(* CODESYS project emCoSys, 3.3.1.1 (IMACS GmbH).library
   Description: Driver for connecting an emBRICK®-LocalMaster via TCP/IP or RS485 over the Modbus LargeBlock Protokoll.
   Author: IMACS GmbH
   Version: 3.3.1.1
   CompiledLibraryCompatibilityVersion: CODESYS V3.5 SP16 Patch 4
   Company: IMACS GmbH
   Title: emCoSys
   LanguageModelAttribute: qualified-access-only
   DefaultNamespace: TPL

Project tree, tasks and I/O mapping:
  CODESYS_Control_Win_V3 : CODESYS Control Win V3, 3S - Smart Software Solutions GmbH, version 3.5.16.40
    application Application
      libraries: SysCom, 3.5.15.0 (System); SysTypes2 Interfaces, * (System)
  libraries: SysMem, * (System); SysCpuHandling, * (System); IoDrvBase, * (System); IoStandard, * (System); IoDriver Parameter Interfaces, * (System); Base Interfaces, * (System); IoDriver Interfaces, * (System); BASIC, 3.31 (OSCAT); CAA Memory, 3.5.12.0 (CAA Technical Workgroup); CAA Types Extern, 3.5.13.0 (CAA Technical Workgroup); Standard, 3.5.15.0 (System); SysSocket, 3.5.15.0 (System); CAA SerialCom, 3.5.15.0 (CAA Technical Workgroup); SysTypes2 Interfaces, * (System); CmpErrors2 Interfaces, * (System)
  function block emCoSys [ST]: IoDrvWriteParameter, IoDrvReadParameter, IoDrvReadInputs, IoDrvIdentify, IoDrvUpdateConfiguration, IoDrvWatchdogTrigger, IoDrvScanModules, IoDrvUpdateMapping, IoDrvWriteOutputs, IoDrvStartBusCycle, IoDrvGetModuleDiagnosis, QueryInterface, FB_Reinit, Initialize, FB_Exit, FB_Init, IoDrvGetConnector, init, connecting, connectionTimedOut, sendInitRq, recvInitRq, receiveData, sendData, closeSocket, initConnection, GetInitializationData, getVars, CRCModbus
  data type emBRICKData
  data type emBRICKMaster
  data type emBRICKSlave
  data type STATES
  data type COM_TYPES
*)

// emBRICKData
TYPE emBRICKData :
STRUCT
	numOfSlaves : BYTE := 0;
	slaves : ARRAY[0..31] OF emBRICKSlave;
	master : emBRICKMaster;
	localMasterAddress : STRING;
	localMasterPort : UINT;
	pRxData : POINTER TO ARRAY[0..252] OF BYTE;
	pTxData : POINTER TO ARRAY[0..252] OF BYTE;
END_STRUCT
END_TYPE

// emBRICKMaster
TYPE emBRICKMaster :
STRUCT
	ID : WORD := 0;
	protocolVersion : BYTE := 0;
	version : BYTE := 0;
	masterType : BYTE := 0;
	uartType : WORD := 0;	
END_STRUCT
END_TYPE

// emBRICKSlave
TYPE emBRICKSlave :
STRUCT
	status : BYTE := 0;
	dataLengthMOSI : BYTE := 0;
	dataLengthMISO : BYTE := 0;
	offsetMOSI : BYTE := 0;
	offsetMISO : BYTE := 0;
	protocolVersion : BYTE := 0;
	moduleVersion : BYTE := 0;
	deviceID : UINT := 0;
	manufacturerID : UINT := 0;
END_STRUCT
END_TYPE

// STATES
TYPE STATES :
(
	GET_VARS := 0,
	INIT := 1,
	CONNECTING := 2,
	SEND_INIT_RQ := 3,
	RECV_INIT_RQ := 4,
	EXCHANGE_DATA := 5,
	CLOSE_SOCKET := 6,
	SEND_DATA := 7,
	RECV_DATA := 8
);
END_TYPE

// COM_TYPES
TYPE COM_TYPES :
(
	ETHERNET := 1,
	RS485 := 2
);
END_TYPE

// emCoSys
{attribute 'symbol':='readwrite'}
FUNCTION_BLOCK emCoSys EXTENDS IoDrvBase IMPLEMENTS ICmpIoDrvParameter
VAR_INPUT
END_VAR
VAR_OUTPUT
	State : STATES := STATES.GET_VARS;
	xCom1OpenError : BOOL;
	xCom1CloseError : BOOL;
	xCom1WriteError : BOOL;
	xCom1ReadError : BOOL;
END_VAR
VAR
	// Application Variables
	SearchArraySendData: ARRAY[0..5] OF BYTE;
	SearchArraySendDataWithCRC: ARRAY[0..7] OF BYTE;

	RECIEVE_DATA_MISSED_RESPONSES: UDINT;
	SEND_DATA_MISSED_RESPONSES: UDINT;
	COM_Type : COM_TYPES;

	ComType : UDINT;
	IP : UDINT;
	ComPort : UDINT;
	Baudrate : UDINT;
	ModbusSlave : UDINT;
	masterOffset : UINT := 448;
		
	// CONSTANTS
	CONNECTIONTIMEOUT_LIMIT : UINT := 500;
	TASKREPETITIONRATE : UINT := 10;
	
	// emBRICK Data
	ebData : emBRICKData;
	pEbData : POINTER TO emBRICKData := ADR(ebData);
	
	// Helpers
	diFlags : DINT;
	ConnectionTimeout : UINT := 0;
	activate : INT := 1;
	fb_Init_Flag : BOOL := FALSE;
		
	// RS485 VARS
	aCom1Params : ARRAY [1..7] OF COM.PARAMETER;
	como1 : COM.Open;
	comc1 : COM.Close;
	comw1 : COM.Write;
	comr1 : COM.Read;

	CRCInit: ARRAY [0..1] OF BYTE;
	CRCInitCompare: ARRAY [0..1] OF BYTE;
	CRCRead: ARRAY [0..1] OF BYTE;
	CRCReadCompare: ARRAY [0..1] OF BYTE;
	RecievedInitMsg: ARRAY[0..252] OF BYTE;
	RecievedSerialMsg: ARRAY[0..252] OF BYTE;
	bufferSerial: ARRAY[0..254] OF BYTE;
	bufferSerialWithCRC: ARRAY[0..254] OF BYTE;
	bufferReadAnswerSerial: ARRAY[0..32000] OF BYTE;
	bufferReadAnswerSerialReceiveData: ARRAY[0..254] OF BYTE;
	bufferReadAnswerSerialSendData: ARRAY[0..254] OF BYTE;
	GetInitializationDataSerial : ARRAY[1..5] OF BYTE := [16#04, 16#10, 16#00, 16#00, 16#7D];
	SearchArrayDynamic : ARRAY[0..2] OF BYTE;
	SearchArray : ARRAY[0..2] OF BYTE;
	ValidateAnswerFromReadArray : ARRAY [0..5] OF BYTE;
	ValidateAnswerFromReadArrayWithCRC  : ARRAY [0..7] OF BYTE;
	CompareBytesInt: UINT;
	CompareBytesIntInit: UINT;
	CaseIntData: INT := 0;
	CaseIntDataRec: INT := 0;
	CaseIntInit: INT := 0;
	RecieveBytesGelesen: __UXINT;
	SendBytesGelesen: __UXINT;
	
	// ETHERNET VARS
	serverAdress : SOCKADDRESS;
	pServerAdress : POINTER TO SOCKADDRESS := ADR(serverAdress);
	buffer : ARRAY[0..511] OF BYTE;
	pBuffer : POINTER TO ARRAY[0..511] OF BYTE := ADR(buffer);
	msgGetInitializationData : ARRAY[0..5] OF BYTE := [16#06, 16#00, 16#02, 16#00, 16#00, 16#00];
	sentBytes : DINT := 0;
	receivedBytes : DINT := 0;
	NUMOFRXBYTES : INT := 506;
	NUMOFTXBYTES : INT := 506;
	socketID : RTS_IEC_HANDLE;
	pResult : POINTER TO RTS_IEC_RESULT;
	connectionEstablished: RTS_IEC_RESULT;
	socketSet : SOCKET_FD_SET;
	socketTimeout : SOCKET_TIMEVAL;

	// Visualization variables
	lampe : BOOL := 0;
	schalter : BOOL := 0;
	cnt : DWORD := 0;
	
	
	_byInputs : ARRAY [0..IOSize-1] OF BYTE;
	_byOutputs : ARRAY [0..IOSize-1] OF BYTE;
	_IIoDrv : ICmpIoDrv;
	_IIoDrvParameter : ICmpIoDrvParameter;
	_xBackGroundDiagStarted : BOOL;
	_bDeactivated : BOOL;
END_VAR
VAR CONSTANT
	CLASSID_CCmpIoDrvTemplate : DWORD := 16#0000FF02;
	IOSize : DWORD := 512;
	m_ciMaxInputs : DWORD := 10; // max nr of parameters to search for in each connector
	m_ciMaxOutputs : DWORD := 10; // max nr of parameters to search for in each connector
	m_ciInputParameterIdStart : DWORD := 1000; // was UDINT
	m_ciOutputParameterIdStart : DWORD := 2000;	// was UDINT
END_VAR

METHOD IoDrvWriteParameter : UDINT
VAR_INPUT
	pConnector : POINTER TO IoConfigConnector;
	pParameter : POINTER TO IoConfigParameter;
	pData : POINTER TO BYTE;
	dwBitSize : DWORD;
	dwBitOffset : DWORD;
END_VAR
VAR
	pParam : POINTER TO IoConfigParameter;
	pstDiagString : POINTER TO STRING;
END_VAR
IF pConnector = 0 OR pParameter = 0 OR pData = 0 THEN
	IoDrvWriteParameter := Errors.ERR_PARAMETER;
	RETURN;	
END_IF

//If IoDrvWriteParameter returns a value unequal ERR_OK, write parameter will be handled by the IO-manager!
//Note: Code must be only implemented here if there are special things to do.

IoDrvWriteParameter := Errors.ERR_OK;

CASE pParameter^.dwParameterId OF
	393221: //simulate diag
		IF pData^ <> 0 THEN
			//set diag string
			pParam := IoMgrConfigGetParameter(pConnector, 4711);
			IF pParam <> 0 THEN
				pstDiagString := IoMgrConfigGetParameterValuePointer(pParam, 0);
				IF pstDiagString <> 0 THEN
					pstDiagString^ := 'Error pending';
				END_IF
			END_IF
			//set diagnostic available flag
			IoMgrConfigSetDiagnosis(pConnector, Connectorflags.CF_CONNECTOR_DIAGNOSTIC_AVAILABLE);
		END_IF
		RETURN;
	393222, 393223:
		//here you can add some special code for the three paraneters
		SysMemCpy((pParameter^.dwValue + dwBitOffset/8), pData, MIN(DWORD_TO_BYTE(dwBitSize/8), UINT_TO_BYTE(pParameter^.wLen / 8)));			
		RETURN;
	4712: //Diag Acknowledge
		IoMgrConfigResetDiagnosis(pConnector, Connectorflags.CF_CONNECTOR_DIAGNOSTIC_AVAILABLE);
		RETURN;
	ELSE
		SysMemCpy(pDest := pParameter^.dwValue + dwBitOffset/8, pSrc := pData, pParameter^.wLen / 8);
END_CASE

IoDrvWriteParameter := Errors.ERR_FAILED;
END_METHOD

METHOD IoDrvReadParameter : UDINT
VAR_INPUT
	pConnector : POINTER TO IoConfigConnector;
	pParameter : POINTER TO IoConfigParameter;
	pData : POINTER TO BYTE;
	dwBitSize : DWORD;
	dwBitOffset : DWORD;
END_VAR
VAR
END_VAR
IF 	pConnector = 0 OR pParameter = 0 OR pData = 0 THEN
	IoDrvReadParameter := Errors.ERR_PARAMETER;
	RETURN;	
END_IF

IoDrvReadParameter := Errors.ERR_OK;

CASE pParameter^.dwParameterId OF
	4711: (* Diag Parameter *)
		IF pParameter^.wLen >= dwBitOffset + dwBitSize THEN 
			SysMemCpy(pData, (pParameter^.dwValue + dwBitOffset/8), MIN(DWORD_TO_BYTE(dwBitSize/8), UINT_TO_BYTE(pParameter^.wLen / 8)));			
			RETURN;
		END_IF
	ELSE
		SysMemCpy(pData, pParameter^.dwValue + dwBitOffset/8, pParameter^.wLen / 8);
END_CASE

// All standard parameters of our device are handled by the IO-manager!
IoDrvReadParameter := Errors.ERR_FAILED;
END_METHOD

METHOD IoDrvReadInputs : UDINT
VAR_INPUT
	pConnectorMapList : POINTER TO IoConfigConnectorMap;
	nCount : DINT;
END_VAR
VAR
	i,j : DINT;
	wSize : WORD;
	pbyIecAddress : POINTER TO BYTE;
	bySrcValue : BYTE;
	bySrcMask : BYTE;
	wSrcIndex : WORD;	
	wDestIndex : WORD;	
END_VAR
IoDrvReadInputs_Count := IoDrvReadInputs_Count + 1;

IF pConnectorMapList = 0 OR nCount = 0 THEN
	IoDrvReadInputs := Errors.ERR_PARAMETER;
	RETURN;
END_IF

FOR i:=0 TO nCount - 1 DO
	IF (pConnectorMapList[i].dwNumOfChannels = 0) THEN
		CONTINUE;
	END_IF
	FOR j:= 0 TO UDINT_TO_UINT(pConnectorMapList[i].dwNumOfChannels) - 1 DO
		//pConnectorMapList[i].pChannelMapList[j].pParameter^.dwDriverSpecific;
		// input medium byteorder: Little Endian:		
		//IoMgrCopyInputLE(ADR(pConnectorMapList[i].pChannelMapList[j]),pConnectorMapList[i].pChannelMapList[j].pParameter^.dwDriverSpecific);
		
		// input medium byteorder: Big Endian:		
		IoMgrCopyInputBE(ADR(pConnectorMapList[i].pChannelMapList[j]),pConnectorMapList[i].pChannelMapList[j].pParameter^.dwDriverSpecific);
		
	END_FOR
END_FOR

IoDrvReadInputs := Errors.ERR_OK;
END_METHOD

{attribute 'conditionalshow' := 'IoDrvDebug'}
METHOD IoDrvIdentify : UDINT
VAR_INPUT
	pConnector : POINTER TO IoConfigConnector;	
END_VAR
VAR
END_VAR
IoDrvIdentify_Count := IoDrvIdentify_Count + 1;
IoDrvIdentify := Errors.ERR_NOTIMPLEMENTED;
END_METHOD


METHOD IoDrvUpdateConfiguration : UDINT
VAR_INPUT
	pConnectorList : POINTER TO IoConfigConnector;
	nCount : DINT;
END_VAR
VAR
	pParameter : POINTER TO IoConfigParameter;	
	pChild : POINTER TO IoConfigConnector;	
	pstConnectorVendorName : POINTER TO STRING;
	pstConnectorDeviceName : POINTER TO STRING;
	dwTest : POINTER TO DWORD;
	Result : RTS_IEC_RESULT;
	iByteoffsetIn : WORD;
	iByteoffsetOut : WORD;	
	i : DWORD;//INT;
	pByte : POINTER TO BYTE;
	pWord : POINTER TO WORD;
	ST_is_a_very_limited_and_dumb_language : STRING;
	bitsPerByte : WORD := 8;
END_VAR
IoDrvUpdateConfiguration_Count := IoDrvUpdateConfiguration_Count + 1;
IoDrvUpdateConfiguration := Errors.ERR_OK;

IF (pConnectorList = 0) THEN
	// Reset application
	// TODO: Free ressources
	RETURN;
END_IF

m_pConnector := IoMgrConfigGetConnector(pConnectorList, ADR(nCount), m_wModuleType, m_dwInstance);

IF m_pConnector = 0 THEN
	IoDrvUpdateConfiguration := ERRORS.ERR_PARAMETER;
	RETURN;
END_IF

//check if device is enabled in the device tree
IF (m_pConnector^.dwFlags AND ConnectorFlags.CF_ENABLE) = 0 THEN
	_bDeactivated := TRUE;
	IoDrvUpdateConfiguration := Errors.ERR_OK;
	RETURN;
END_IF

IF m_pConnector^.hIoDrv = 0 THEN
	m_pConnector^.hIoDrv := m_hInterface;
	m_pConnector^.pFather^.hIoDrv := m_hInterface;
	
	{IF defined (pou:IoMgrConfigSetDiagnosis)}
	IoMgrConfigSetDiagnosis(m_pConnector,
							ConnectorFlags.CF_DRIVER_AVAILABLE OR
							ConnectorFlags.CF_CONNECTOR_FOUND OR
							ConnectorFlags.CF_CONNECTOR_CONFIGURED OR
							ConnectorFlags.CF_CONNECTOR_ACTIVE);
	{END_IF}
	
	{IF defined (pou:IoMgrConfigSetDiagnosis)}
	IoMgrConfigSetDiagnosis(m_pConnector^.pFather,
							ConnectorFlags.CF_DRIVER_AVAILABLE OR
							ConnectorFlags.CF_CONNECTOR_FOUND OR
							ConnectorFlags.CF_CONNECTOR_CONFIGURED OR
							ConnectorFlags.CF_CONNECTOR_ACTIVE);
	{END_IF}

	{IF defined (pou:IoMgrSetDriverProperties)}			
		IoMgrSetDriverProperties(m_hInterface, DRVPROP_CONSISTENCY OR DRVPROP_BACKGROUND_GETDIAG);
		//Note: background diagnosis property flag is optional (supported with 3.5.1.0 runtime)
	{END_IF}										

	//Read some parameters
	pParameter := IoMgrConfigGetParameter(m_pConnector, 393218);
	IF pParameter <> 0 THEN
		pstConnectorVendorName := IoMgrConfigGetParameterValuePointer(pParameter, ADR(Result));
	END_IF
	pParameter := IoMgrConfigGetParameter(m_pConnector, 393219);
	IF pParameter <> 0 THEN
		pstConnectorDeviceName := IoMgrConfigGetParameterValuePointer(pParameter, ADR(Result));
	END_IF
	pParameter := IoMgrConfigGetParameter(m_pConnector, 393220);	(* test parameter *)
	IF (pParameter <> 0) THEN
		dwTest := IoMgrConfigGetParameterValueDword(pParameter, ADR(Result));	(* Test parameter value *)			
	END_IF

	iByteoffsetIn := 0;
	iByteOffsetOut := 0;
	//Go through all childs of the device
	pChild := IoMgrConfigGetFirstChild(m_pConnector, ADR(nCount), m_pConnector);
	WHILE (pChild <> 0) DO
		IF (pChild^.dwFlags AND ConnectorFlags.CF_ENABLE) <> 0 THEN
			pChild^.hIoDrv := m_hInterface;	
			{IF defined (pou:IoMgrConfigSetDiagnosis)}
			IoMgrConfigSetDiagnosis(pChild,
									ConnectorFlags.CF_DRIVER_AVAILABLE OR
									ConnectorFlags.CF_CONNECTOR_FOUND OR
									ConnectorFlags.CF_CONNECTOR_CONFIGURED OR
									ConnectorFlags.CF_CONNECTOR_ACTIVE);
			{END_IF}

			// Setup Config Data
			
			//pEbData^.slaves[slaveCounter].dataLengthMOSI;				// number of Bytes received by the Slave
			//pEbData^.slaves[slaveCounter].dataLengthMISO;				// number of Bytes sent by the Slave
			//pEbData^.slaves[slaveCounter].protocolVersion;				// highest possible protocol version this Slave is able to receive
			//pEbData^.slaves[slaveCounter].moduleVersion;				// Version number of the Slave itself
			//pEbData^.slaves[slaveCounter].deviceID;		// ID of the Slave
											
			//pEbData^.slaves[slaveCounter].manufacturerID;		// Manufacturer of the Slave
														
			//pEbData^.slaves[slaveCounter].offsetMOSI;			// Offset in the txBuffer for Data sent to the Slave
			//pEbData^.slaves[slaveCounter].offsetMISO;			// Offset in the rxBuffer for Data sent to the Slave
			
			//Setup I/O area
			FOR i := 0 TO m_ciMaxInputs DO
				pParameter := IoMgrConfigGetParameter(pChild, m_ciInputParameterIdStart + i);		(* inputs *)
				IF (pParameter <> 0) THEN
					pParameter^.dwDriverSpecific := ADR(_byInputs[iByteoffsetIn]);  							
					iByteoffsetIn := iByteoffsetIn + (pParameter^.wLen / bitsPerByte);							
				END_IF
			END_FOR
			
			FOR i := 0 TO m_ciMaxOutputs DO
				pParameter := IoMgrConfigGetParameter(pChild, m_ciOutputParameterIdStart + i);		(* outputs *)
				IF (pParameter <> 0) THEN
					pParameter^.dwDriverSpecific := ADR(_byOutputs[iByteoffsetOut]);  							
					iByteoffsetOut := iByteoffsetOut + (pParameter^.wLen / bitsPerByte);							
				END_IF
			END_FOR
		END_IF
		pChild := IoMgrConfigGetNextChild(pChild, ADR(nCount), m_pConnector);
	END_WHILE
END_IF
END_METHOD

{attribute 'conditionalshow' := 'IoDrvDebug'}
METHOD IoDrvWatchdogTrigger : UDINT
VAR_INPUT
	pConnector : POINTER TO IoConfigConnector;	
END_VAR
VAR
END_VAR
IoDrvWatchdogTrigger_Count := IoDrvWatchdogTrigger_Count + 1;
IoDrvWatchdogTrigger := Errors.ERR_OK;
END_METHOD

{attribute 'conditionalshow' := 'IoDrvDebug'}
METHOD IoDrvScanModules : UDINT
VAR_INPUT
	pConnector : POINTER TO IoConfigConnector;
	ppConnectorList : POINTER TO POINTER TO IoConfigConnector;
	pnCount : POINTER TO DINT;	
END_VAR
VAR
END_VAR
IoDrvScanModules_Count := IoDrvScanModules_Count + 1;
IoDrvScanModules := Errors.ERR_NOTIMPLEMENTED;
END_METHOD

{attribute 'conditionalshow' := 'IoDrvDebug'}
METHOD IoDrvUpdateMapping : UDINT
VAR_INPUT
	pTaskMapList : POINTER TO IoConfigTaskMap;
	nCount : DINT;	
END_VAR
VAR
END_VAR
IoDrvUpdateMapping_Count := IoDrvUpdateMapping_Count + 1;

IF (pTaskMapList = 0) THEN
	IoDrvUpdateMapping := Errors.ERR_PARAMETER;
	RETURN;
END_IF

IoDrvUpdateMapping := Errors.ERR_OK;
END_METHOD

METHOD IoDrvWriteOutputs : UDINT
VAR_INPUT
	pConnectorMapList : POINTER TO IoConfigConnectorMap;
	nCount : DINT;
END_VAR
VAR
	i,j : DINT;
	wSize : WORD;
	pbyIecAddress : POINTER TO BYTE;
	bySrcValue : BYTE;
	wSrcIndex : WORD;	
	bySrcMask : BYTE;
	wDestIndex : WORD;	
END_VAR
IoDrvWriteOutputs_Count := IoDrvWriteOutputs_Count + 1;

IF pConnectorMapList = 0 OR nCount = 0 THEN
	IoDrvWriteOutputs := Errors.ERR_PARAMETER;
	RETURN;
END_IF

FOR i:=0 TO nCount - 1 DO
	IF (pConnectorMapList[i].dwNumOfChannels = 0) THEN
		CONTINUE;
	END_IF
	FOR j:= 0 TO UDINT_TO_UINT(pConnectorMapList[i].dwNumOfChannels) - 1 DO
		// output medium byteorder: Little Endian:		
		//IoMgrCopyOutputLE(ADR(pConnectorMapList[i].pChannelMapList[j]),pConnectorMapList[i].pChannelMapList[j].pParameter^.dwDriverSpecific);
		
		// output medium byteorder: Big Endian:		
		IoMgrCopyOutputBE(ADR(pConnectorMapList[i].pChannelMapList[j]),pConnectorMapList[i].pChannelMapList[j].pParameter^.dwDriverSpecific);
	END_FOR
END_FOR

IoDrvWriteOutputs := Errors.ERR_OK;
END_METHOD

//{attribute 'conditionalshow' := 'IoDrvDebug'}
METHOD IoDrvStartBusCycle : UDINT
VAR_INPUT
	pConnector : POINTER TO IoConfigConnector;
END_VAR
VAR
	
END_VAR
IoDrvStartBusCycle_Count := IoDrvStartBusCycle_Count + 1;

//if background diagnosis is not active call IoDrvGetModuleDiagnosis; normally it will be called by the runtime if DRVPROP_BACKGROUND_GETDIAG is set
IF NOT _xBackGroundDiagStarted THEN
	IoDrvGetModuleDiagnosis(m_pConnector); //DRVPROP_BACKGROUND_GETDIAG not set or runtime version < V3.5.1.0
END_IF

//optional: call IoDrvWatchdogTrigger or set driver property DRVPROP_WATCHDOG in UpdateConfiguration
IoDrvWatchdogTrigger(pConnector);

IoDrvStartBusCycle := Errors.ERR_OK;

CASE State OF
	STATES.GET_VARS:
		getVars();
		IF getVars() = TRUE THEN
			State := STATES.INIT;
		END_IF


	(* not connected - Try to open socket and connect *)
	STATES.INIT:
		init();
		State := STATES.CONNECTING;
		
	
	(* wait for the socket to connect to the server *)
	STATES.CONNECTING:
		// Check if a connection Timeout occured
		IF connectionTimedOut() = TRUE THEN
			State := STATES.CLOSE_SOCKET;
		END_IF
		// Connect to Server; Count State up on success and configure socket
		IF connecting() = TRUE THEN
			ConnectionTimeout := 0;
			sentBytes := 0;
			// Continue to next State
			State := STATES.SEND_INIT_RQ;
		ELSE
			ConnectionTimeout := ConnectionTimeout + TASKREPETITIONRATE;		
		END_IF;
		
	(* Request emBRICK Initialization Data from Localmaster *)
	STATES.SEND_INIT_RQ: 
		/// Check if a connection Timeout occured
		IF connectionTimedOut() = TRUE THEN
			State := STATES.CLOSE_SOCKET;
		END_IF
		// send frame, continue on success
		IF sendInitRq() = TRUE THEN
			// Count State up
			State := STATES.RECV_INIT_RQ;
			receivedBytes := 0;
			ConnectionTimeout := 0;
		ELSE // count timeout up
			ConnectionTimeout := ConnectionTimeout + TASKREPETITIONRATE;
		END_IF
			
	(* Receive Initialization Data *)		
	STATES.RECV_INIT_RQ: 
		// Check if a connection Timeout occured
		IF connectionTimedOut() = TRUE THEN
			State := STATES.CLOSE_SOCKET;
		END_IF
		// receive frame and continue on success
		IF recvInitRq() = TRUE THEN
			// Count State up
			sentBytes := 0;
			ConnectionTimeout := 0;
			State := STATES.EXCHANGE_DATA;
		ELSE // count timeout up
			ConnectionTimeout := ConnectionTimeout + TASKREPETITIONRATE;	
		END_IF
	(* Exchange Data with Localmaster *)	
	STATES.EXCHANGE_DATA:
		// Check if a connection Timeout occured
		IF connectionTimedOut() = TRUE THEN
			State := STATES.CLOSE_SOCKET;
		END_IF
		// receive Data sent from Localmaster
		IF receiveData() = TRUE THEN
			sentBytes := 0;
			ConnectionTimeout := 0;
		ELSE
			ConnectionTimeout := ConnectionTimeout + TASKREPETITIONRATE;		
		END_IF;
		// send Data to Localmaster 
		IF sendData() = TRUE THEN
			receivedBytes := 0;
		ELSE
			ConnectionTimeout := ConnectionTimeout + TASKREPETITIONRATE;
		END_IF	
	(* Close Socket -> Back to Case 1 *)	
	STATES.CLOSE_SOCKET: 
		closeSocket();
		// return to Init State
		State := STATES.INIT;
END_CASE
END_METHOD

METHOD IoDrvGetModuleDiagnosis : UDINT
VAR_INPUT
	pConnector : POINTER TO IoConfigConnector;
END_VAR
VAR
END_VAR
IF pConnector = 0 THEN
	//we are called from the background task
	_xBackGroundDiagStarted := TRUE;
END_IF

//Todo: update connectorflags if something changed

IoDrvGetModuleDiagnosis_Count := IoDrvGetModuleDiagnosis_Count + 1;
IoDrvGetModuleDiagnosis := Errors.ERR_NOTIMPLEMENTED;
END_METHOD

METHOD QueryInterface : POINTER TO POINTER TO BYTE
VAR_INPUT
	iid : DWORD; (* InterfaceID *)
	pResult : POINTER TO UDINT;	
END_VAR
VAR
END_VAR
QueryInterface_Count := QueryInterface_Count + 1;
IF iid = ITFID_ICmpIoDrv THEN
	QueryInterface := ADR(_IIoDrv);
	AddRef();
	IF (pResult <> 0) THEN
		pResult^ := Errors.ERR_OK;
	END_IF
	RETURN;	
ELSIF iid = ITFID_ICmpIoDrvParameter THEN
	QueryInterface := ADR(_IIoDrvParameter);
	AddRef();
	IF (pResult <> 0) THEN
		pResult^ := Errors.ERR_OK;
	END_IF	
	RETURN;	
ELSE
	QueryInterface := SUPER^.QueryInterface(iid, pResult);
END_IF
END_METHOD

{attribute 'conditionalshow' := 'IoDrvDebug'}
METHOD FB_Reinit : BOOL
VAR_INPUT
END_VAR
VAR
END_VAR
FB_Reinit_Count := FB_Reinit_Count + 1;
FB_Reinit := TRUE;
END_METHOD

{attribute 'conditionalshow' := 'IoDrvDebug'}
METHOD Initialize : UDINT
VAR_INPUT
	wModuleType : UINT;
	dwInstance : UDINT;
	pConnector : POINTER TO IoConfigConnector; 
END_VAR
VAR
END_VAR
Initialize_Count := Initialize_Count + 1;

m_wModuleType := wModuleType;
m_dwInstance := dwInstance;
m_Info.wModuleType := wModuleType;

Initialize := Errors.ERR_OK;
END_METHOD

{attribute 'conditionalshow' := 'IoDrvDebug'}
METHOD FB_Exit : BOOL
VAR_INPUT
	bInCopyCode: BOOL;	
END_VAR
VAR
	// Helper
END_VAR
FB_Exit_Count := FB_Exit_Count + 1; //Taskcounter
FB_Exit := TRUE;
END_METHOD

METHOD FB_Init : BOOL
VAR_INPUT
	bInitRetains: BOOL;
	bInCopyCode: BOOL;
END_VAR
VAR
	Result : UDINT;
	
	// Helper
	finishedFBInit : BOOL := FALSE;
END_VAR
FB_Init_Count := FB_Init_Count + 1;

// from CoDeSys
m_Info.szDriverName := 'IoDrvTemplateIEC';
m_Info.szVendorName := 'MyCompany';
m_Info.szDeviceName := 'MyCard';
m_Info.wModuleType := 40100;

_IIoDrv := THIS^;
_IIoDrvParameter := THIS^;

m_IBaseItf := THIS^;
m_hInterface := IoMgrRegisterInstance2(CLASSID_CCmpIoDrvTemplate, m_IBaseItf, ADR(Result));

IF initConnection() = TRUE THEN
	FB_Init := TRUE;	
	fb_Init_Flag := TRUE;
END_IF
END_METHOD

METHOD IoDrvGetConnector : POINTER TO IoConfigConnector
VAR_INPUT
	pResult : POINTER TO RTS_IEC_RESULT;
END_VAR
VAR
END_VAR
IF m_pConnector = 0 THEN
	IF pResult <> 0 THEN
		pResult^ := Errors.ERR_FAILED;
	END_IF
	IoDrvGetConnector := 0;	
	RETURN;
END_IF
IF pResult <> 0 THEN
	pResult^ := Errors.ERR_OK;
END_IF
IoDrvGetConnector := m_pConnector;
END_METHOD

METHOD init
VAR_INPUT
END_VAR
VAR
	pParameter: POINTER TO IoConfigParameter;
	Result : RTS_IEC_RESULT;
	pLocalMasterIP : POINTER TO STRING;
	pLocalComPort : POINTER TO UDINT;
	pLocalBaudrate : POINTER TO UDINT;
END_VAR
// Set pointer to rx, tx-Buffer
ebData.pRxData := ADR(_byInputs);
ebData.pTxData := ADR(_byOutputs);

CASE COM_Type OF
	COM_TYPES.ETHERNET:
		// Initialize SOCKADRESS-Struct and set Pointer
		serverAdress.sin_addr.ulAddr := IP;							// set IP to connect to
		serverAdress.sin_family := SOCKET_AF_INET;					// TCP/IP
		serverAdress.sin_port := SysSockHtons(7086);				// set Socket of Server to connect to
		pServerAdress := ADR(serverAdress);							// set Pointer to variable holding server data
		
		// Open Socket
		socketID := SysSockCreate(SOCKET_AF_INET, SOCKET_STREAM, SOCKET_IPPROTO_IP, pResult);
		
		// Configure Socket as nonblocking
		SysSockIoctl(hSocket:= socketID, diCommand:= SOCKET_FIONBIO, pdiParameter:= ADR(activate));
		
		// Add Socket to socket set
		SysSockFdInit(socketID, socketSet);
		
		// Init Timeout struct
		socketTimeout.tv_usec := 500000;
		
		// Connect to LocalMaster as Client
		SysSockConnect(socketID, pServerAdress, SIZEOF(serverAdress));	
		
		// wait for connect
		ConnectionTimeout := 0;
		
	COM_TYPES.RS485:
		// Initialize COM Port
		//The parameters are set for the COM Port
		aCom1Params[1].udiParameterId := COM.CAA_Parameter_Constants.udiPort;
		aCom1Params[1].udiValue := ComPort; // the correct Port should be adapted
		aCom1Params[2].udiParameterId := COM.CAA_Parameter_Constants.udiBaudrate;
		aCom1Params[2].udiValue := Baudrate;
		aCom1Params[3].udiParameterId := COM.CAA_Parameter_Constants.udiParity;
		aCom1Params[3].udiValue := INT_TO_UDINT(COM.PARITY.NONE);
		aCom1Params[4].udiParameterId := COM.CAA_Parameter_Constants.udiStopBits;
		aCom1Params[4].udiValue := INT_TO_UDINT(COM.STOPBIT.ONESTOPBIT);
		aCom1Params[5].udiParameterId := COM.CAA_Parameter_Constants.udiTimeout;
		aCom1Params[5].udiValue := 0;
		aCom1Params[6].udiParameterId := COM.CAA_Parameter_Constants.udiByteSize;
		aCom1Params[6].udiValue := 8;
		aCom1Params[7].udiParameterId := COM.CAA_Parameter_Constants.udiBinary;
		aCom1Params[7].udiValue := 0;
		
		//The first Port is opened with the given parameters
		como1(xExecute := TRUE, usiListLength:=SIZEOF(aCom1Params)/SIZEOF(COM.PARAMETER),pParameterList:= ADR(aCom1Params));
		//COM Port
		IF como1.xError THEN
			como1(xExecute := FALSE);
			xCom1OpenError := TRUE;
		END_IF
		
		IF como1.xDone THEN
			xCom1OpenError := FALSE;
		END_IF
END_CASE
END_METHOD

METHOD connecting : BOOL
VAR_INPUT
END_VAR
CASE COM_Type OF
	COM_TYPES.ETHERNET:
		// Check Socket
		connectionEstablished := SysSockSelect(diWidth:= 1, pfdRead:= ADR(socketSet), pfdWrite := ADR(socketSet), pfdExcept := ADR(socketSet), ptvTimeout:= ADR(socketTimeout), pdiReady:= ADR(activate) );	
		IF connectionEstablished = 0 THEN
			connecting := TRUE;	
		ELSE
			connecting := FALSE;
		END_IF
		
	COM_TYPES.RS485:
		connecting := TRUE;
END_CASE
END_METHOD

METHOD connectionTimedOut : BOOL
VAR_INPUT
END_VAR
IF ConnectionTimeout >= CONNECTIONTIMEOUT_LIMIT THEN
	connectionTimedOut := TRUE;	
ELSE
	connectionTimedOut := FALSE;	
END_IF
END_METHOD

METHOD sendInitRq : BOOL
VAR_INPUT
END_VAR
VAR
	CRC :DWORD;
END_VAR
CASE COM_Type OF
	COM_TYPES.ETHERNET:
		// send frame, count sent Bytes up
		sentBytes := sentBytes + SysSockSend(hSocket:= socketID, pbyBuffer:= ADR(msgGetInitializationData), SIZEOF(msgGetInitializationData), diFlags:= diFlags, pResult:= pResult);
		// Check if all Bytes have been sent
		IF sentBytes >= SIZEOF(msgGetInitializationData) THEN
			SendInitRq := TRUE;
		ELSE
			SendInitRq := FALSE;
		END_IF
		
	COM_TYPES.RS485:
		CASE CaseIntInit OF
			0:
			// send Data to Localmaster over serial
			// prepare frame
			_BUFFER_CLEAR(PT:=ADR(bufferSerial) , SIZE:=SIZEOF(bufferSerial) );
			_BUFFER_CLEAR(PT:=ADR(bufferSerialWithCRC) , SIZE:=SIZEOF(bufferSerialWithCRC) );
			bufferSerial[0] := UDINT_TO_BYTE(ModbusSlave);	// Slave Number
			// load BUSData into buffer
			sysmemcpy(ADR(bufferSerial[1]), ADR(GetInitializationDataSerial), SIZEOF(GetInitializationDataSerial));// load bytes of txBuffer into buffer
			// Calc CRC
			CRC:= CRCModbus(CRC_DATA:=ADR(bufferSerial) , CRC_SIZE:= UINT_TO_INT(1+SIZEOF(GetInitializationDataSerial)));
			sysmemcpy(ADR(bufferSerialWithCRC), ADR(bufferSerial), SIZEOF(bufferSerial));
			sysmemcpy(ADR(bufferSerialWithCRC[1+SIZEOF(GetInitializationDataSerial)]), ADR(CRC), SIZEOF(CRC));						// Add calc CRC
			// send frame
			// Write COM PORT
			comw1(xExecute := TRUE,hCom:= como1.hCom,pBuffer:= ADR(bufferSerialWithCRC),szSize:= 1+SIZEOF(GetInitializationDataSerial)+2);	// write COM
				// success
				IF comw1.xDone THEN
					comw1(xExecute:= FALSE);
					CaseIntInit := 1;	
				END_IF
				IF comw1.xError THEN
					comw1(xExecute:= FALSE);
				END_IF
			1:
			comr1(xExecute := TRUE,hCom:= como1.hCom, pBuffer:= ADR(bufferReadAnswerSerial), szBuffer:= SIZEOF(bufferReadAnswerSerial));
			IF comr1.xDone THEN
				//Build Search Array
				SearchArray[0] := UDINT_TO_BYTE(ModbusSlave);
				SearchArray[1] := 16#04;
				SearchArray[2] := 16#FA;
				//Check for expectet Bytes in recieved Bytes
				CompareBytesIntInit := INT_TO_UINT(BUFFER_COMP( 
					PT1:= ADR(bufferReadAnswerSerial), 
					SIZE1:= UINT_TO_INT(SIZEOF(bufferReadAnswerSerial)), 
					PT2:= ADR(SearchArray), 
					SIZE2:= UINT_TO_INT(SIZEOF(SearchArray)), 
					START:= 0));
				IF CompareBytesIntInit <> 16#FFFF THEN
					sysmemcpy(ADR(RecievedInitMsg), ADR(bufferReadAnswerSerial[CompareBytesIntInit]), 252);
					sysmemcpy(ADR(CRCInit), ADR(bufferReadAnswerSerial[CompareBytesIntInit+253]), 2);
					// Calc and compare CRC
					CRC:= CRCModbus(CRC_DATA:=ADR(RecievedInitMsg) , CRC_SIZE:= UINT_TO_INT(SIZEOF(RecievedInitMsg)));
					sysmemcpy(ADR(CRCInitCompare), ADR(CRC), SIZEOF(CRC));
					CompareBytesIntInit := INT_TO_UINT(BUFFER_COMP( 
						PT1:= ADR(CRCInit), 
						SIZE1:= UINT_TO_INT(SIZEOF(CRCInit)), 
						PT2:= ADR(CRCInitCompare), 
						SIZE2:= UINT_TO_INT(SIZEOF(CRCInitCompare)), 
						START:= 0));
					IF CompareBytesIntInit = 0 THEN
						// Store received Data to Struct						
						GetInitializationData(peBData := ADR(ebData));
						sendInitRq := TRUE;
					END_IF
				END_IF
				comr1(xExecute:= FALSE);	// Reset xExecute Flag
				CaseIntInit := 0;
			END_IF
			IF comr1.xError THEN
				comr1(xExecute:= FALSE);
				CaseIntInit := 0;
			END_IF
		END_CASE
END_CASE
END_METHOD

METHOD recvInitRq : BOOL
VAR_INPUT
END_VAR

VAR
	x: INT;
END_VAR
CASE COM_Type OF
	COM_TYPES.ETHERNET:
		// receive frame and count received Bytes up
		receivedBytes := receivedBytes + SysSockRecv(hSocket:= socketID, pbyBuffer:= pBuffer, diBufferSize:= SIZEOF(buffer), diFlags:= diFlags, pResult:= pResult);
		// Check if all bytes have been received
		IF receivedBytes >= 6 THEN
			// if all bytes have been received, copy buffer into rxData
			sysmemcpy(ebData.pRxData, pBuffer, SIZEOF(buffer));
			// Store received Data to Struct
			GetInitializationData(peBData := ADR(ebData));
			RecvInitRq :=  TRUE;
		ELSE
			RecvInitRq := FALSE;
		END_IF
		
	COM_TYPES.RS485:
		recvInitRq :=  TRUE;
END_CASE
END_METHOD

METHOD receiveData : BOOL
VAR_INPUT
END_VAR
VAR
	CRC :DWORD;
	i : UINT;
	MOSI : BYTE;
	MISO : BYTE;
	CRCCompareInt: UINT;
	FoundInt: INT;
END_VAR
CASE COM_Type OF
	COM_TYPES.ETHERNET:
		// receive Data sent from Localmaster
		receivedBytes := receivedBytes + SysSockRecv(hSocket:= socketID,	pbyBuffer:= pBuffer, diBufferSize:= SIZEOF(buffer), diFlags:= diFlags, pResult:= pResult);
		IF receivedBytes >= 6 THEN
			// for now, only receive the actually useful information
			sysmemcpy(ebData.pRxData, ADR(buffer[8]), receivedBytes-8);
			// TODO receive Master Data and Offset
			receiveData := TRUE;
		ELSE
			receiveData := FALSE;
		END_IF
		
	COM_TYPES.RS485:
		CASE CaseIntDataRec OF
			0:
			// send Data to Localmaster over serial
			// prepare frame
			_BUFFER_CLEAR(PT:=ADR(bufferSerial) , SIZE:=SIZEOF(bufferSerial) );
			_BUFFER_CLEAR(PT:=ADR(bufferSerialWithCRC) , SIZE:=SIZEOF(bufferSerialWithCRC) );
			bufferSerial[0] := UDINT_TO_BYTE(ModbusSlave);	// Slave Number	6
			bufferSerial[1] := 16#17;	// Function Code	7
			bufferSerial[2] := 16#00;	// Memory Read Start Address	8 
			bufferSerial[3] := 16#00;	// Memory Read Start Address 	9
			bufferSerial[4] := 16#00;	// Read Quantity	10
			//Calc quantity
			MISO := 0;
			FOR i := 0 TO (pEbData^.numOfSlaves) BY 1 DO
				MISO := MISO + pEbData^.slaves[i].dataLengthMISO;
			END_FOR
			IF MISO.0 = 1 THEN
				MISO:=MISO+1;
			END_IF						
			bufferSerial[5] := MISO/2;	// Read Quantity 	11
			//Change SearchArray to Quanitiy of MISO	
			SearchArray[0] := UDINT_TO_BYTE(ModbusSlave);	// Slave Number 
			SearchArray[1] := 16#17;	// Function Code 
			SearchArray[2] := MISO;	// Quantity 
			
			bufferSerial[6] := 16#00;	// Memory Write Start Address  12
			bufferSerial[7] := 16#00;	// Memory Write Start Address	13	
			bufferSerial[8] := 16#00;	// Write Quantity 	14
			//Calc quantity
			MOSI := 0;
			FOR i := 0 TO (pEbData^.numOfSlaves) BY 1 DO
				MOSI := MOSI + pEbData^.slaves[i].dataLengthMOSI;				// number of Bytes received by the Slave
			END_FOR
			bufferSerial[9] := MOSI;	// Quantity 15
			bufferSerial[10] := MOSI*2;	// ByteSize <- Didn't use	16
			// load BUSData into buffer
			sysmemcpy(ADR(bufferSerial[11]), ebData.pTxData, (MOSI*2));// load bytes of txBuffer into buffer
			// Calc CRC
			CRC:= CRCModbus(CRC_DATA:=ADR(bufferSerial) , CRC_SIZE:= UINT_TO_INT(11+(MOSI*2)));
			sysmemcpy(ADR(bufferSerialWithCRC), ADR(bufferSerial), SIZEOF(bufferSerial));
			sysmemcpy(ADR(bufferSerialWithCRC[11+(MOSI*2)]), ADR(CRC), SIZEOF(CRC));						// Add calc CRC
			// send frame
			//Prepare ValidateAnswerFromReadArray
			sysmemcpy(ADR(ValidateAnswerFromReadArray), ADR(bufferSerialWithCRC), (6));// load bytes of txBuffer into buffer
			// Calc CRC
			CRC:= CRCModbus(CRC_DATA:=ADR(ValidateAnswerFromReadArray) , CRC_SIZE:= UINT_TO_INT(SIZEOF(ValidateAnswerFromReadArray)));
			sysmemcpy(ADR(ValidateAnswerFromReadArrayWithCRC), ADR(ValidateAnswerFromReadArray), SIZEOF(ValidateAnswerFromReadArray));
			sysmemcpy(ADR(ValidateAnswerFromReadArrayWithCRC[6]), ADR(CRC), SIZEOF(CRC));	
			// Write COM PORT
			comw1(xExecute := TRUE,hCom:= como1.hCom,pBuffer:= ADR(bufferSerialWithCRC),szSize:= 11+(MOSI*2)+2);
						IF comw1.xDone THEN
							RECIEVE_DATA_MISSED_RESPONSES:= RECIEVE_DATA_MISSED_RESPONSES+1;
							comw1(xExecute:= FALSE);	// Reset xExecute Flag
							CaseIntDataRec:=1;
						END_IF
						IF comw1.xError THEN
							comw1(xExecute:= FALSE);
							CaseIntDataRec:=1;
						END_IF
		1:
		//Read the response from the request
		comr1(xExecute := TRUE,hCom:= como1.hCom, pBuffer:= ADR(bufferReadAnswerSerial), szBuffer:= SIZEOF(bufferReadAnswerSerial), szSize=>RecieveBytesGelesen);
			IF comr1.xDone THEN
				comr1(xExecute:= FALSE);
				//Check for expectet Bytes in recieved Bytes
				FoundInt := INT_TO_UINT(BUFFER_COMP( 
					PT1:= ADR(bufferReadAnswerSerial), 
					SIZE1:= SIZEOF(bufferReadAnswerSerial), 
					PT2:= ADR(SearchArray), 
					SIZE2:= SIZEOF(SearchArray), 
					START:= 0));
				// If expectet Bytes are found copy the recieved Data to pRxData
					sysmemcpy(ADR(RecievedSerialMsg), ADR(bufferReadAnswerSerial[FoundInt]), 3+SearchArray[2]);
					sysmemcpy(ADR(CRCRead), ADR(bufferReadAnswerSerial[FoundInt+3+SearchArray[2]]), 2);
					// Calc and compare CRC
					CRC:= CRCModbus(CRC_DATA:=ADR(RecievedSerialMsg) , CRC_SIZE:= 3+SearchArray[2]);
					sysmemcpy(ADR(CRCReadCompare), ADR(CRC), SIZEOF(CRC));
					CRCCompareInt := INT_TO_UINT(BUFFER_COMP( 
						PT1:= ADR(CRCRead), 
						SIZE1:= UINT_TO_INT(SIZEOF(CRCRead)), 
						PT2:= ADR(CRCReadCompare), 
						SIZE2:= UINT_TO_INT(SIZEOF(CRCReadCompare)), 
						START:= 0));
					IF CRCCompareInt = 0 THEN
						RECIEVE_DATA_MISSED_RESPONSES:= RECIEVE_DATA_MISSED_RESPONSES-1;
						sysmemcpy(ebData.pRxData, ADR(bufferReadAnswerSerial[FoundInt+3]), SearchArray[2]);
						receiveData :=  TRUE;
					END_IF
				comr1(xExecute:= FALSE);	// Reset xExecute Flag
				CaseIntInit := 0;
			END_IF
			IF comr1.xError THEN
						comr1(xExecute:= FALSE);
					END_IF
				CaseIntDataRec:=0;
		END_CASE
END_CASE
END_METHOD

METHOD sendData : BOOL
VAR_INPUT
END_VAR
VAR
	CRC :DWORD;
	i : UINT;
	MOSI : BYTE;
	MISO : BYTE;
	CRCCompareInt: UINT;
	FoundInt: INT;
END_VAR
CASE COM_Type OF
	COM_TYPES.ETHERNET:
		// send Data to Localmaster 
		NUMOFTXBYTES := 506;
		// prepare frame
		buffer[0] := WORD_TO_BYTE(NUMOFTXBYTES MOD 256);//16#FA;//	// LSB number of Bytes the slave is supposed to receive
		buffer[1] := WORD_TO_BYTE(NUMOFTXBYTES / 256);//16#01;//	// MSB number of Bytes the slave is supposed to receive 
		buffer[2] := 16#10;	// command byte - exchange Data
		buffer[3] := 0;
		buffer[4] := 0;
		buffer[5] := 0;	
		sysmemcpy(ADR(buffer[6]), ADR(masterOffset), SIZEOF(masterOffset));		// Copy master Offset into Bytes 3 and 4
		// TODO load Master Data
		// load BUSData into buffer
		sysmemcpy(ADR(buffer[8]), ebData.pTxData, 500);						// load 500 bytes of txBuffer into buffer
		// send frame
		sentBytes := sentBytes + SysSockSend(hSocket:= socketID, pbyBuffer:= pBuffer, NUMOFTXBYTES, diFlags:= diFlags, pResult:= pResult);
		// check if all bytes were sent 
		IF sentBytes >= NUMOFTXBYTES THEN
			sendData := TRUE;
		ELSE
			sendData := FALSE;
		END_IF
	COM_TYPES.RS485:
		CASE CaseIntData OF
			0:
			CaseIntData:=1;
			1:
			CaseIntData:=0;
			sendData := TRUE;
		END_CASE
END_CASE
END_METHOD

METHOD closeSocket : BOOL
VAR_INPUT
END_VAR
CASE COM_Type OF
	COM_TYPES.ETHERNET:
		// Clear socket set
		socketSet.fd_array[0] := 0;
		socketSet.fd_count := 0;
		// Close Socket
		SysSockClose(hSocket:= socketID);
		
	COM_TYPES.RS485:
		//Close Com Port
		comc1(xExecute := TRUE, hCom:= como1.hCom);
		IF comc1.xError THEN
			xCom1CloseError := TRUE;
		END_IF
		IF como1.xError THEN
			como1.xExecute := FALSE;
		END_IF
END_CASE
END_METHOD

METHOD initConnection : BOOL
VAR_INPUT
END_VAR
	CASE State OF
		STATES.GET_VARS:
		// get User Vars from devdesc.xml
			getVars();
			IF getVars() = TRUE THEN
				State := STATES.INIT;
			END_IF
		STATES.INIT:
			// init ethernet
			init();
			// Connect to Server
			State := STATES.CONNECTING;
			// reset init_flag
			fb_Init_Flag := FALSE;
			
			// Open Connection
			(* wait for the socket to connect to the server *)
		STATES.CONNECTING:
			// Check if a connection Timeout occured
			IF connectionTimedOut() = TRUE THEN
				State := STATES.CLOSE_SOCKET;
			END_IF
			// Connect to Server; Count State up on success and configure socket
			IF connecting() = TRUE THEN
				ConnectionTimeout := 0;
				sentBytes := 0;
				// Continue to next State
				State := STATES.SEND_INIT_RQ;
			ELSE
				ConnectionTimeout := ConnectionTimeout + TASKREPETITIONRATE;		
			END_IF;
			
		(* Request emBRICK Initialization Data from Localmaster *)
		STATES.SEND_INIT_RQ: 
			/// Check if a connection Timeout occured
			IF connectionTimedOut() = TRUE THEN
				State := STATES.CLOSE_SOCKET;
			END_IF
			// send frame, continue on success
			IF sendInitRq() = TRUE THEN
				// Count State up
				State := STATES.RECV_INIT_RQ;
				receivedBytes := 0;
				ConnectionTimeout := 0;
			ELSE // count timeout up
				ConnectionTimeout := ConnectionTimeout + TASKREPETITIONRATE;		
			END_IF
				
		(* Receive Initialization Data *)		
		STATES.RECV_INIT_RQ: 
			// Check if a connection Timeout occured
			IF connectionTimedOut() = TRUE THEN
				State := STATES.CLOSE_SOCKET;
			END_IF
			// receive frame and continue on success
			IF recvInitRq() = TRUE THEN
				// Count State up
				sentBytes := 0;
				ConnectionTimeout := 0;
				State := STATES.EXCHANGE_DATA;
				// End Initialization
				initConnection := TRUE;
			ELSE // count timeout up
				ConnectionTimeout := ConnectionTimeout + TASKREPETITIONRATE;	
			END_IF
			
		(* Close Socket -> Back to Case 1 *)	
		STATES.CLOSE_SOCKET: 
			closeSocket();
			// return to Init State
			State := STATES.INIT;
	
	END_CASE
END_METHOD

METHOD GetInitializationData : INT
VAR_INPUT
	pEbData : POINTER TO emBRICKData;
END_VAR
VAR
	i : UINT;
	sizeOfStruct : UINT := (SIZEOF(emBRICKSlave) - 1);
	buffer : ARRAY[0..511] OF BYTE;
	pParameter: POINTER TO IoConfigParameter;
	Result : INT;
	pByte : POINTER TO BYTE;
	pWord : POINTER TO WORD;
	pString : POINTER TO STRING;
	sVar : STRING;
	pChild : POINTER TO IoConfigConnector;
	nCount : DINT := 6;
END_VAR
(* store boardBUS settings *)
CASE COM_Type OF
	COM_TYPES.ETHERNET:
		sysmemcpy(ADR(buffer), pEbData^.pRxData + 6, receivedBytes - 6);
	COM_TYPES.RS485:
		sysmemcpy(ADR(buffer), ADR(RecievedInitMsg[3]), SIZEOF(RecievedInitMsg)-3);
END_CASE


// Number of Slaves
pEbData^.numOfSlaves 				:= buffer[0];									
pParameter := IoMgrConfigGetParameter(m_pConnector, 400002);
IF (pParameter <> 0) THEN
	pByte := IoMgrConfigGetParameterValuePointer(pParameter, ADR(Result));	
END_IF
pByte^ := pEbData^.numOfSlaves;

// Local-Master ID
pEbData^.master.ID 				:= (buffer[2] * 256) + buffer[3];			
pParameter := IoMgrConfigGetParameter(m_pConnector, 400003);
IF (pParameter <> 0) THEN
	pWord := IoMgrConfigGetParameterValuePointer(pParameter, ADR(Result));		
END_IF
pWord^ := pEbData^.master.ID;

CASE pEbData^.master.ID OF
	1601: sVar := 'Z-LWCS-M32-01 - All Features';	
	1602: sVar := 'Z-LWCS-M32-02 - All Features except WLAN';
	1603: sVar := 'Z-LWCS-M32-03 - Only LAN';
	1604: sVar := 'Z-LWCS-M32-04 - Only RSxx, CAN';
	1611: sVar := 'Z-PatBridgeMX-11 - LAN, RSxx, CAN';
	1612: sVar := 'Z-PatBridgeMX-12 - Only LAN';
	1613: sVar := 'Z-UniBridgeMX-13 RB - LAN, WLAN, CAN, RSxx';
	1614: sVar := 'Z-UniBridgeMX-14 RB - Only LAN';
ELSE
	sVar := 'Unknown Module';
END_CASE

pParameter := IoMgrConfigGetParameter(m_pConnector, 393219);
IF pParameter <> 0 THEN
	pString := IoMgrConfigGetParameterValuePointer(pParameter, ADR(Result));
END_IF
pString^:= sVar;

// Local Master Version
pEbData^.master.version 			:= buffer[5];		
pParameter := IoMgrConfigGetParameter(m_pConnector, 400004);
IF (pParameter <> 0) THEN
	pByte := IoMgrConfigGetParameterValuePointer(pParameter, ADR(Result));		
END_IF
pByte^ := pEbData^.master.version;

// Local-/Remote-Master Version
pEbData^.master.protocolVersion 			:= buffer[4];		
pParameter := IoMgrConfigGetParameter(m_pConnector, 400005);
IF (pParameter <> 0) THEN
	pByte := IoMgrConfigGetParameterValuePointer(pParameter, ADR(Result));		
END_IF
pByte^ := pEbData^.master.protocolVersion;

// Local-Master Manufacturer ID
pEbData^.master.masterType 			:= buffer[6];		
pParameter := IoMgrConfigGetParameter(m_pConnector, 400006);
IF (pParameter <> 0) THEN
	pByte := IoMgrConfigGetParameterValuePointer(pParameter, ADR(Result));		
END_IF
pByte^ := pEbData^.master.masterType;

CASE pEbData^.master.masterType OF
	1: sVar := 'IMACS GmbH';
ELSE
	sVar := 'Unknown Manufacturer';
END_CASE

pParameter := IoMgrConfigGetParameter(m_pConnector, 393218);
IF pParameter <> 0 THEN
	pString := IoMgrConfigGetParameterValuePointer(pParameter, ADR(Result));
END_IF
pString^:= sVar;

// Local-Master Periphery
pEbData^.master.uartType 			:= (buffer[7] * 256) + buffer[8];		
pParameter := IoMgrConfigGetParameter(m_pConnector, 400007);
IF (pParameter <> 0) THEN
	pWord := IoMgrConfigGetParameterValuePointer(pParameter, ADR(Result));		
END_IF
pWord^ := pEbData^.master.uartType;

// do not store bus_status as of now, as it does not hold any valuable information at this point

pChild := IoMgrConfigGetFirstChild(m_pConnector, ADR(nCount), m_pConnector);

(* store Slave Information *)

FOR i := 0 TO (pEbData^.numOfSlaves) BY 1 DO
	pEbData^.slaves[i].status 			:= buffer[ (i*sizeOfStruct) + 1 + 8 ];				// actual Status of Slave
	pEbData^.slaves[i].dataLengthMOSI 	:= buffer[ (i*sizeOfStruct) + 2 + 8 ];				// number of Bytes received by the Slave
	pEbData^.slaves[i].dataLengthMISO 	:= buffer[ (i*sizeOfStruct) + 3 + 8 ];				// number of Bytes sent by the Slave
	pEbData^.slaves[i].protocolVersion 	:= buffer[ (i*sizeOfStruct) + 4 + 8 ];				// highest possible protocol version this Slave is able to receive
	pEbData^.slaves[i].moduleVersion 	:= buffer[ (i*sizeOfStruct) + 5 + 8 ];				// Version number of the Slave itself
	pEbData^.slaves[i].deviceID 		:= (buffer[ (i*sizeOfStruct) + 6 + 8 ] * 256)		// ID of the Slave
										+	buffer[ (i*sizeOfStruct) + 7 + 8 ];	
	pEbData^.slaves[i].manufacturerID 	:= (buffer[ (i*sizeOfStruct) + 8 + 8 ] * 256)		// Manufacturer of the Slave
										+	buffer[ (i*sizeOfStruct) + 9 + 8 ];		
	pEbData^.slaves[i].offsetMOSI	 	:= buffer[ (i*sizeOfStruct) + 10 + 8 ];			// Offset in the txBuffer for Data sent to the Slave
	pEbData^.slaves[i].offsetMISO	 	:= buffer[ (i*sizeOfStruct) + 11 + 8 ];			// Offset in the rxBuffer for Data sent to the Slave
	
	// Device ID
	pParameter := IoMgrConfigGetParameter(pChild, 400002);
	IF pParameter <> 0 THEN
		pWord := IoMgrConfigGetParameterValuePointer(pParameter, ADR(Result));
		IF pWord <> 0 THEN
			pWord^:= pEbData^.slaves[i].deviceID;				// Device ID of the emBRICK®-module
		END_IF
	END_IF
	
	// Data Length Out
	pParameter := IoMgrConfigGetParameter(pChild, 400003);
	IF pParameter <> 0 THEN
		pByte := IoMgrConfigGetParameterValuePointer(pParameter, ADR(Result));
		IF pByte <> 0 THEN
			pByte^:= pEbData^.slaves[i].dataLengthMOSI;				// number of Bytes received by the Slave
		END_IF
	END_IF
	
	// Data Length In
	pParameter := IoMgrConfigGetParameter(pChild, 400004);
	IF pParameter <> 0 THEN
		pByte := IoMgrConfigGetParameterValuePointer(pParameter, ADR(Result));
		IF pByte <> 0 THEN
			pByte^:= pEbData^.slaves[i].dataLengthMISO;				// number of Bytes sent by the Slave
		END_IF
	END_IF
	
	// Protocol Version
	pParameter := IoMgrConfigGetParameter(pChild, 400005);
	IF pParameter <> 0 THEN
		pByte := IoMgrConfigGetParameterValuePointer(pParameter, ADR(Result));
		IF pByte <> 0 THEN
			pByte^:= pEbData^.slaves[i].protocolVersion;				// Implemented emBRICK® Protocol-Version of the module
		END_IF
	END_IF
	
	// Hardware Version
	pParameter := IoMgrConfigGetParameter(pChild, 400006);
	IF pParameter <> 0 THEN
		pByte := IoMgrConfigGetParameterValuePointer(pParameter, ADR(Result));
		IF pByte <> 0 THEN
			pByte^:= pEbData^.slaves[i].moduleVersion;				// Hardware Version of the emBRICK®-module
		END_IF
	END_IF
	
	// Manufacturer ID
	pParameter := IoMgrConfigGetParameter(pChild, 400007);
	IF pParameter <> 0 THEN
		pWord := IoMgrConfigGetParameterValuePointer(pParameter, ADR(Result));
		IF pWord <> 0 THEN
			pWord^:= pEbData^.slaves[i].manufacturerID;				// Device ID of the emBRICK®-module
		END_IF
	END_IF
	
	// Data Offset Out
	pParameter := IoMgrConfigGetParameter(pChild, 400008);
	IF pParameter <> 0 THEN
		pByte := IoMgrConfigGetParameterValuePointer(pParameter, ADR(Result));
		IF pByte <> 0 THEN
			pByte^:= pEbData^.slaves[i].offsetMOSI;				// Offset of Data Area(MOSI)
		END_IF
	END_IF
	
	// Data Offset In
	pParameter := IoMgrConfigGetParameter(pChild, 400009);
	IF pParameter <> 0 THEN
		pByte := IoMgrConfigGetParameterValuePointer(pParameter, ADR(Result));
		IF pByte <> 0 THEN
			pByte^:= pEbData^.slaves[i].offsetMISO;				// Offset of Data Area(MISO)
		END_IF
	END_IF
	
	// get next child
	pChild := IoMgrConfigGetNextChild(pChild, ADR(nCount), m_pConnector);
END_FOR
END_METHOD

METHOD getVars : BOOL
VAR_INPUT
END_VAR
VAR
	pParameter: POINTER TO IoConfigParameter;
	Result : RTS_IEC_RESULT;
	pLocalComType : POINTER TO UDINT;
	pLocalMasterIP : POINTER TO STRING;
	pLocalComPort : POINTER TO UDINT;
	pLocalBaudrate : POINTER TO UDINT;
	pLocalModbusSlave : POINTER TO UDINT;
END_VAR
// Get COM-Type
pParameter := IoMgrConfigGetParameter(m_pConnector, 399996);
IF pParameter <> 0 THEN
	pLocalComType := IoMgrConfigGetParameterValuePointer(pParameter, ADR(Result));
	ComType := pLocalComType^;
END_IF

// Get Modbus Slave Address
pParameter := IoMgrConfigGetParameter(m_pConnector, 399997);
IF pParameter <> 0 THEN
	pLocalModbusSlave := IoMgrConfigGetParameterValuePointer(pParameter, ADR(Result));
	ModbusSlave := pLocalModbusSlave^;
END_IF

// Get TCP/IP-Adress
pParameter := IoMgrConfigGetParameter(m_pConnector, 400001);
IF pParameter <> 0 THEN
	pLocalMasterIP := IoMgrConfigGetParameterValuePointer(pParameter, ADR(Result));
	SysSockInetAddr(pLocalMasterIP^,ADR(IP));					// generate IP to connect to from String
END_IF

// Get COM Port
pParameter := IoMgrConfigGetParameter(m_pConnector, 399998);
IF pParameter <> 0 THEN
	pLocalComPort := IoMgrConfigGetParameterValuePointer(pParameter, ADR(Result));
	ComPort := pLocalComPort^;
END_IF

// Get COM Baudrate
pParameter := IoMgrConfigGetParameter(m_pConnector, 399999);
IF pParameter <> 0 THEN
	pLocalBaudrate := IoMgrConfigGetParameterValuePointer(pParameter, ADR(Result));
	Baudrate := pLocalBaudrate^;
END_IF

IF ComType = 1 THEN
	COM_Type := COM_TYPES.ETHERNET;
	IF 	IP > 0 THEN
		getVars := TRUE;
	END_IF	
END_IF

IF ComType = 2 THEN
	COM_Type := COM_TYPES.RS485;
	State := STATES.SEND_INIT_RQ;
	IF 	ComPort > 0 THEN
		getVars := TRUE;
	END_IF	
END_IF
END_METHOD

METHOD CRCModbus : DWORD
VAR_INPUT
	CRC_DATA: POINTER TO ARRAY[0..32000] OF BYTE;
	CRC_SIZE: INT;
END_VAR
CRCModbus := CRC_GEN(
	PT:= CRC_DATA,
	SIZE:= CRC_SIZE,
	PL:= 16,
	PN:= 16#8005,
	INIT:= 16#FFFF,
	REV_IN:= TRUE, 
	REV_OUT:= TRUE,
	XOR_OUT:= 0);
END_METHOD

END_FUNCTION_BLOCK
